PROGRAM p08_counter
VAR
	counter: CTUD;
	S0: BOOL;
	S1: BOOL;
	S2: BOOL;
	S3: BOOL;
	value: WORD;
END_VAR

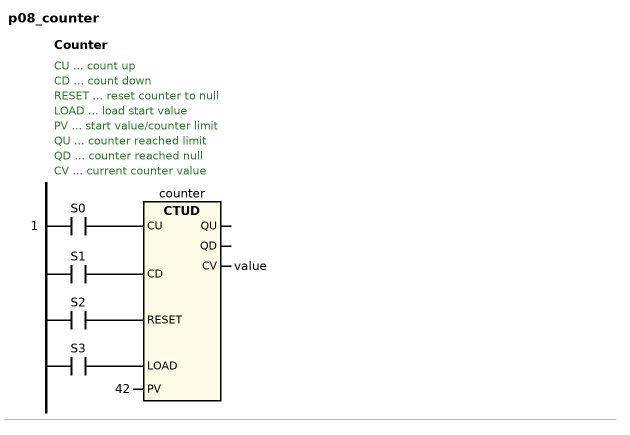
// NETWORK 1: Counter
// CU ... count up
// CD ... count down
// RESET ... reset counter to null
// LOAD ... load start value
// PV ... start value/counter limit
// QU ... counter reached limit
// QD ... counter reached null
// CV ... current counter value
counter(CU := S0, CD := S1, RESET := S2, LOAD := S3, PV := 42, CV => value); // CTUD

END_PROGRAM

(* stored: Version 1.1.0.1, ProductVersion 3.1.4024.13
   POU p08_counter: Id {5b80c4c7-148d-416b-9cf3-bb59d285eea0}, SpecialFunc None *)
